TYPE
    DUT_MsgToAmsPortHeader :
    STRUCT
        nServiceCode : UDINT;
        nClassId : UDINT;
        nInstanceId : UDINT;
        nAttributeId : UDINT;
        nReservedId : UDINT;
        nGeneralStatus : UDINT;
        nAdditionalStatus : UDINT;
        nDataLen : UDINT;
    END_STRUCT
END_TYPE

(* stored: Version 1.1.0.1, ProductVersion 3.1.4024.12
   DUT DUT_MsgToAmsPortHeader: Id {dcb19c93-a31a-4949-8397-00a83c3b92d2} *)
